FUNCTION_BLOCK Rotativo (* Template for a Basic Function Block Type *)
  (* Standard: 61499-2 *)
  (* Version 1.0, 2025-02-05, Bruno *)
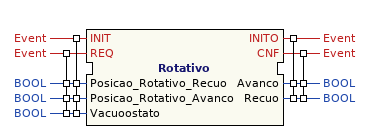
  EVENT_INPUT
    INIT WITH Posicao_Rotativo_Recuo, Posicao_Rotativo_Avanco, Vacuoostato; (* Initialization Request *)
    REQ WITH Posicao_Rotativo_Recuo, Posicao_Rotativo_Avanco, Vacuoostato; (* Normal Execution Request *)
  END_EVENT
  EVENT_OUTPUT
    INITO WITH Avanco, Recuo; (* Initialization Confirm *)
    CNF WITH Avanco, Recuo; (* Execution Confirmation *)
  END_EVENT
  VAR_INPUT
    Posicao_Rotativo_Recuo : BOOL; (* Input event qualifier *)
    Posicao_Rotativo_Avanco : BOOL;
    Vacuoostato : BOOL;
  END_VAR
  VAR_OUTPUT
    Avanco : BOOL; (* Output event qualifier *)
    Recuo : BOOL;
  END_VAR
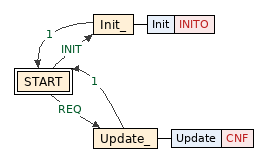
  EC_STATES
    START; (* Initial State *)
    Init_ : Init -> INITO;
    Update_ : Update -> CNF;
  END_STATES
  EC_TRANSITIONS
    START TO Init_ := INIT;
    Init_ TO START := 1;
    START TO Update_ := REQ;
    Update_ TO START := 1;
  END_TRANSITIONS
  ALGORITHM Init IN ST:
Avanco:=FALSE;
Recuo:=FALSE;
  END_ALGORITHM
  ALGORITHM Update IN ST:
IF Posicao_Rotativo_Recuo AND Vacuoostato THEN

Avanco:=TRUE;
Recuo:=FALSE;

END_IF;

IF Posicao_Rotativo_Avanco AND (NOT Vacuoostato) THEN

Recuo:=TRUE;
Avanco:=FALSE;

END_IF;
  END_ALGORITHM
END_FUNCTION_BLOCK
